(* PLC project turret, Dassault Systèmes ControlBuild 2024x *)
(* stored: creationDateTime 2023-10-03T11:13:44-01:00 *)

FUNCTION_BLOCK drill.turret
  VAR_INPUT
    speed : REAL := 0.0;
  END_VAR
  VAR_INPUT
    forward : BOOL := false;
    backward : BOOL := false;
    highSpeed : BOOL := false;
    lowSpeed : BOOL := false;
  END_VAR
  VAR_OUTPUT
    axlePosition : REAL := 0.0;
    forwardEnd : BOOL := false;
    forwardDeceleration : BOOL := false;
    backwardDeceleration : BOOL := false;
    backwardEnd : BOOL := false;
  END_VAR
  VAR
    speedIncrement : REAL := 0.0;
  END_VAR
  VAR CONSTANT
    lockingFault : BOOL := false;
    forwardEndFault : BOOL := false;
    forwardEndValue : BOOL := false;
    forwardDecelerationFault : BOOL := false;
    forwardDecelerationValue : BOOL := false;
    backwardDecelerationFault : BOOL := false;
    backwardDecelerationValue : BOOL := false;
    backwardEndFault : BOOL := false;
    backwardEndValue : BOOL := false;
    axleLength : REAL := 100.0;
    forwardDecelerationPosition : DINT := 70;
    backwardDecelerationPosition : DINT := 30;
    range : DINT := 10;
  END_VAR


ACTION C_source_code:
/* Evolution of the axe in function of the input orders		*/
if ( !lockingFault)
{
	speedIncrement = speed * CLOCK_PERIOD / 1000000.0;
	axlePosition += speedIncrement;
	if (axlePosition > axleLength)
		axlePosition = axleLength;

	if (axlePosition < 0.0)
		axlePosition = 0.0;
}


/*Calculation of the sensor states						 */
forwardEnd = (( !forwardEndFault && (axlePosition == axleLength)) || (forwardEndFault &forwardEndValue));
forwardDeceleration = (( !forwardDecelerationFault &&(axlePosition >= forwardDecelerationPosition)&&(axlePosition <= (forwardDecelerationPosition + range))) || (forwardDecelerationFault && forwardDecelerationValue));
backwardDeceleration = (( !backwardDecelerationFault && (axlePosition >= backwardDecelerationPosition) & (axlePosition <= (backwardDecelerationPosition + range))) || (backwardDecelerationFault && backwardDecelerationValue));
backwardEnd = (( !backwardEndFault && (axlePosition == 0)) || (backwardEndFault &backwardEndValue));
END_ACTION
END_FUNCTION_BLOCK
